{attribute 'linkalways'} 
{attribute 'no_explicit_call' := 'This FB is a CLASS and must be accessed using methods or properties'}
{attribute 'enable_dynamic_creation'}
FUNCTION_BLOCK FINAL ADD_UDINT EXTENDS Node
VAR
	in1 : _UDINT(0);
	in2 : _UDINT(0);
	out : _UDINT(0);
END_VAR

METHOD PUBLIC Clone : I_Node
VAR
	pNode : POINTER TO ADD_UDINT;
END_VAR
pNode := __NEW(ADD_UDINT);
Clone := pNode^;
END_METHOD

METHOD FB_init : BOOL
VAR_INPUT
	bInitRetains : BOOL; // if TRUE, the retain variables are initialized (warm start / cold start)
	bInCopyCode : BOOL;  // if TRUE, the instance afterwards gets moved into the copy code (online change)
END_VAR
AddInput('in1',THIS^.in1);
AddInput('in2',THIS^.in2);
AddOutput('out', THIS^.out);
END_METHOD

METHOD PROTECTED OnExecute
VAR
END_VAR
out.Value := in1.Value + in2.Value;
END_METHOD

END_FUNCTION_BLOCK

(* stored: Version 1.1.0.1, ProductVersion 3.1.4024.15
   POU ADD_UDINT: Id {5cb835b0-8be3-4154-84fd-7d5f5b1851a9}, SpecialFunc None
   Folder Constructor: Id {fe70b8dc-b270-4548-8e67-9595f6fb96be}
   Method Clone: Id {e95e8099-c753-42cc-8594-f6d914b4af72}
   Method FB_init: Id {1d90716f-5cdc-4961-9a7e-f197077b3a5e}
   Method OnExecute: Id {aac1e2bf-af7d-492a-8879-ee1e80cfa84a} *)
